PROGRAM MAIN
VAR
	nCounter	: INT;
END_VAR

nCounter:=nCounter+1;
UN01();
DeviceState();

END_PROGRAM

(* stored: Version 1.1.0.1, ProductVersion 3.1.4024.12
   POU MAIN: Id {70a8f826-1275-472a-9418-f8d98fd0b926}, SpecialFunc None *)
